# EPICS substitutions: ek9000App/Db/EL2024_mbboDirect.substitutions
file EL2024.template
{       pattern
        {
                TERMINAL,

        }
        {
        }
}
